TYPE eSeparationState :
(
	step0 := 0,
	step1 := 1,
	step2 := 2,
	step3 := 3,
	step4 := 4,
	step5 := 5,
	step6 := 6,
	step7 := 7,
	step8 := 8,
	step9 := 9
);
END_TYPE

(* stored: Version 1.1.0.1, ProductVersion 3.1.0.23
   DUT eSeparationState: Id {84a9fcb8-644e-43fe-a3e3-ba06a587011e} *)
